(*
SPDX-FileCopyrightText: © 2026 Oleksandr Tiutyk <trofimich@gmail.com>
SPDX-License-Identifier: MIT
License: https://opensource.org/license/mit
*)

(*!
<summary>Provides a common execution entry point for an object.</summary>
<description>
The caller drives execution; this interface does not schedule calls. Configuration, lifecycle and execution
timing are defined by the concrete object or its specialized interface.
</description>
*)

INTERFACE IExecutable EXTENDS IObject

(*!
<summary>Performs one invocation of the object's execution logic.</summary>
<description>
Returning from this method does not by itself indicate completion of a multi-cycle operation. Required
preparation, call frequency, state changes and exception handling follow the specialized contract. Do not
assume repeated calls within one PLC cycle are equivalent to a single call.
</description>
*)

METHOD Execute
END_METHOD

END_INTERFACE

(* stored: Version 1.1.0.1
   Itf IExecutable: Id {19ad5037-eddf-40c2-bed5-b3c4caabf442}
   Method Execute: Id {929462e9-5c53-48d1-a008-4a9304fa5e51} *)
